PROGRAM prgPV
VAR
	lrPowerPV				: LREAL;				//{#lynus.ag#()}
		// extend or reduce amount of PV Inverters
	lrPowerPV_1				: LREAL;				//{#lynus.ag#()}
	lrPowerPV_2				: LREAL;				//{#lynus.ag#()}
	uint_setPoint_onetenth: UINT;						//{#lynus.ag#()}

	m_shared: BOOL;
END_VAR
VAR PERSISTENT
	lrCounterPV_1				: LREAL;				//{#lynus.ag#()}
	lrCounterPV_2				: LREAL;				//{#lynus.ag#()}
END_VAR

IF m_shared THEN
	prgPV_shared();
	lrPowerPV 				:= prgPV_shared.lrPowerPV;
	lrPowerPV_1 			:= prgPV_shared.lrPowerPV_1;
	lrPowerPV_2 			:= prgPV_shared.lrPowerPV_2;
	uint_setPoint_onetenth 	:= prgPV_shared.uint_setPoint_onetenth;
	lrCounterPV_1			:= prgPV_shared.lrCounterPV_1;
	lrCounterPV_2			:= prgPV_shared.lrCounterPV_2;
ELSE
	prgPV_separate();
	lrPowerPV 				:= prgPV_separate.lrPowerPV;
	lrPowerPV_1 			:= prgPV_separate.lrPowerPV_1;
	lrPowerPV_2 			:= prgPV_separate.lrPowerPV_2;
	uint_setPoint_onetenth 	:= prgPV_separate.uint_setPoint_onetenth;
	lrCounterPV_1			:= prgPV_separate.lrCounterPV_1;
	lrCounterPV_2			:= prgPV_separate.lrCounterPV_2;
END_IF

END_PROGRAM

(* stored: Version 1.1.0.1, ProductVersion 3.1.4024.12
   POU prgPV: Id {ae7d2570-60b2-47cc-af1f-731ca08638e7}, SpecialFunc None *)
